PROGRAM MAIN
VAR
	Machine : FB_Machine; 
	
END_VAR

Machine();

END_PROGRAM

(* stored: Version 1.1.0.1, ProductVersion 3.1.4024.9
   POU MAIN: Id {8cc2debb-a12d-41b6-8e74-bb242da5ef2f}, SpecialFunc None *)
